FUNCTION_BLOCK Insertion //2d insertion that combines a slider (alignment) and screw (push)
VAR_INPUT
	enable : BOOL;
END_VAR
VAR_INPUT //interface references to existing drives
	slider : I_EncodedDrive;
	screw : I_ContinuousDrive;
END_VAR
VAR_OUTPUT
	contact AT %I* : BOOL; //may be removed from this FB and put into a 3rd GVL for floating sensors
	softContact : BOOL; //temporary
	
	active : BOOL;
	error : BOOL;
	home : BOOL;
	
	homingComplete : BOOL;
	
	sliderPos : LREAL;
END_VAR
(*
this FB encapsulates 2 drives into a generic insertion machine
both drives should be declared externally in Hardware GVL as a concrete FB
Insertion instance should be declared and called in module scope, with the drives from Hardware GVL passed in by Interface reference
*)

softContact := slider.contact AND screw.contact; //temporary

homingComplete := (*slider.HomeSet AND*) screw.HomeSet;

active := slider.Busy OR screw.Busy;
error := slider.Error OR screw.Error;
home := slider.AtHome AND screw.AtHome;

sliderPos := slider.CurrentPosition;

METHOD align : BOOL
VAR_INPUT
	targetPos : REAL;
END_VAR
slider.moveAbsolute(newTarget := targetPos);
END_METHOD

METHOD homingSequence : BOOL
VAR_INPUT
END_VAR
IF NOT slider.homeSet THEN
	slider.homingSequence();
END_IF

IF NOT screw.homeSet THEN
	screw.homingSequence();
END_IF

homingSequence := homingComplete;
END_METHOD

METHOD press : BOOL
VAR_INPUT
END_VAR
screw.moveContinuous(direction := MC_Negative_Direction);
END_METHOD

METHOD release : BOOL
VAR_INPUT
END_VAR
screw.moveContinuous(direction := MC_Positive_Direction);
END_METHOD

METHOD reset : BOOL
VAR_INPUT
END_VAR
(*
implementation TBD, drive interfaces currently do not specify a reset method
*)
//slider.reset();
//screw.reset();
END_METHOD

METHOD stop : BOOL
VAR_INPUT
END_VAR
screw.stop();
slider.stop();
END_METHOD

METHOD traverse : BOOL
VAR_INPUT
	direction : MC_Direction;
END_VAR
slider.moveContinuous(direction := MC_Negative_Direction);
END_METHOD

END_FUNCTION_BLOCK

(* stored: Version 1.1.0.1, ProductVersion 3.1.4024.11
   POU Insertion: Id {474cec8b-539b-4b97-8920-b045f392c812}, SpecialFunc None
   Method align: Id {150b5680-ccac-4b88-b9bd-ce3a432e6e4b}
   Method homingSequence: Id {1eff6ad7-4509-4cdc-81af-eef38809ec7f}
   Method press: Id {4b68a98e-5d52-4750-8c51-39e9aab9887f}
   Method release: Id {43664641-2403-4070-8d32-2915d9eeb09e}
   Method reset: Id {e21f4572-1f7b-4ac9-bdab-f9be9f3716fd}
   Method stop: Id {5bc5b53c-ac4b-4bbc-9d14-d47b3c4cd68f}
   Method traverse: Id {2976ba6d-a5c4-4581-84e8-a5c41da415dd} *)
